// TIA Portal V17 export
// export: Created 2025-03-10T13:09:14.3412957Z, ExportSetting WithDefaults, DisplayName Totally Integrated Automation Portal, DisplayVersion V17 Update 8, DisplayName TIA Portal Openness, DisplayVersion V17 Update 8, DisplayName TIA Portal Version Control Interface, DisplayVersion V17, DisplayName SINAMICS Startdrive Advanced, DisplayVersion V17 SP2, DisplayName SINAMICS Startdrive G110M, G120, G120C, G120D, G120P, G115D, DisplayVersion V17 SP2, DisplayName SINAMICS Startdrive G130, G150, S120, S150, SINAMICS MV, S210, DisplayVersion V17 SP2, DisplayName STEP 7 Professional, DisplayVersion V17 Update 8, DisplayName SINUMERIK ONE STEP 7 Toolbox, DisplayVersion V17 Update 12, DisplayName SINUMERIK 840D sl STEP 7 Toolbox, DisplayVersion V17 Update 12, DisplayName STEP 7 Safety, DisplayVersion V17 Update 6, DisplayName WinCC Advanced, DisplayVersion V17 Update 8
DATA_BLOCK "LBP_InternalDB8"   // DB8
TITLE = Internal DB for basic program / DB interno para el programa básico / Interner DB für Grundprogramm
{ S7_Optimized_Access := 'FALSE'; DB_Accessible_From_OPC_UA := 'FALSE' }
AUTHOR : SINUMERIK
FAMILY : SINUMERIK_ONE
VERSION : 6.15
// DB only for internal use in the basic program / DB solo para uso interno en el programa básico / DB nur zur internen Verwendung im Grundprogramm
// stored: AutoNumber false, DBAccessibleFromOPCUA false, DBAccessibleFromWebserver true, IsOnlyStoredInLoadMemory false, IsWriteProtectedInAS false
   VAR RETAIN
      DoNotUse0 : DWord;
      Reserved4 : Array[4..7] of Byte;
      FirstCycle : Byte;   // nicht verwendet / not used / no se utiliza
      InternalUse9_0 : Bool;
      InternalUse9_1 : Bool;
      AL_404031 : Bool;
      InternalUse10 : Array[1..10] of Bool;
      InternalUse12 : SInt;
      InternalUse14 : Array[1..10] of Bool;
      InternalUse16 : SInt;
      InternalUse18 : Array[1..10] of Bool;
      InternalUse20 : Array[1..10] of Bool;
      Reserved22 : Array[22..53] of Byte;   // nicht verwendet / not used / no se utiliza
      InternalUse54 : DWord;
      InternalUse58 : DWord;
      DoNotUse62 : DWord;
      Reserved66 : Array[66..75] of Byte;
      InternalUse76 : DWord;
      InternalUse80 : DInt;   // nur zur internen Verwendung / internal use only / solo para uso interno
      InternalUse84 : LReal;   // nur zur internen Verwendung / internal use only / solo para uso interno
      MinCycleTime : Int;   // nicht verwendet / not used / no se utiliza
      AdaptTime : Int;   // nicht verwendet / not used / no se utiliza
      ActCycleTime : Int;   // nicht verwendet / not used / no se utiliza
      InternalUse98 : HW_ANY;   // nur zur internen Verwendung / internal use only / solo para uso interno
      InternalUse100 : LReal;
   END_VAR
BEGIN
END_DATA_BLOCK
